// TIA Portal V16 export
// export: Created 2025-08-01T13:38:08.397994Z, ExportSetting WithDefaults, DisplayName Totally Integrated Automation Portal, DisplayVersion V16, DisplayName TIA Portal Version Control Interface, DisplayVersion V16, DisplayName TIA Portal Openness, DisplayVersion V16, DisplayName STEP 7 Professional, DisplayVersion V16, DisplayName STEP 7 Safety, DisplayVersion V16, DisplayName WinCC Advanced, DisplayVersion V16
DATA_BLOCK "SCLTestingEnc_DB"   // DB94
VERSION : 0.1
// stored: AutoNumber true, InstanceOfName SCLTestingEnc, InstanceOfType FB
"SCLTestingEnc"
BEGIN
END_DATA_BLOCK
